// TwinCAT 3 PLC project Untitled1
// ProgramVersion: 3.1.4024.0
// libraries:
//   Tc2_MC2, * (Beckhoff Automation GmbH)
//   Tc2_Standard, * (Beckhoff Automation GmbH)
//   Tc2_System, * (Beckhoff Automation GmbH)
//   Tc3_Module, * (Beckhoff Automation GmbH)
// project tree:
//   GVLs/ GVL_Axes.TcGVL
//   / PlcTask.TcTTO
//   POUs/ MAIN.TcPOU (not stored)
// real-time tasks:
//   TASK PlcTask: cycle T#10ms, priority 20, ADS port 350
// motion (NC):
//   TASK NC-Task 1 SAF: cycle T#2ms, priority 4, ADS port 501
//   TASK NC-Task 1 SVB: cycle T#10ms, priority 8, ADS port 511
//   AXIS Axis 1 (id 1)
//     General: UnitName=Degree
//     OtherSettings: AllowMotionCmdToSlave=true
//     encoder EncType=19
//       EncPara: ScaleFactorNumerator=360, ScaleFactorDenominator=16777216, MaxCount=#xffffffff
//     drive DrvType=16
//       DrvPara: MaxCount=#xffffffff, DriveControlDWord=#x00020000
//         Analog: TorqueSetpointScale=10, ScaleFactorActTorque=0.1
//         TimeComp: TaskDelayCycles=1
//     controller CtrType=1
//       CtrPara: PriorControlFactor=1
//         PosDiffControl: Range=5000
//         Observer: BandWidth=20
//   AXIS Axis 2 (id 2)
//     General: UnitName=Degree
//     OtherSettings: AllowMotionCmdToSlave=true
//     encoder EncType=19
//       EncPara: ScaleFactorNumerator=360, ScaleFactorDenominator=16777216, MaxCount=#xffffffff
//     drive DrvType=16
//       DrvPara: MaxCount=#xffffffff, DriveControlDWord=#x00020000
//         Analog: TorqueSetpointScale=10, ScaleFactorActTorque=0.1
//         TimeComp: TaskDelayCycles=1
//     controller CtrType=1
//       CtrPara: PriorControlFactor=1
//         PosDiffControl: Range=5000
//         Observer: BandWidth=20
//   AXIS Axis 3 (id 3)
//     General: UnitName=Degree
//     OtherSettings: AllowMotionCmdToSlave=true
//     encoder EncType=19
//       EncPara: ScaleFactorNumerator=360, ScaleFactorDenominator=16777216, MaxCount=#xffffffff
//     drive DrvType=16
//       DrvPara: MaxCount=#xffffffff, DriveControlDWord=#x00020000
//         Analog: TorqueSetpointScale=10, ScaleFactorActTorque=0.1
//         TimeComp: TaskDelayCycles=1
//     controller CtrType=1
//       CtrPara: PriorControlFactor=1
//         PosDiffControl: Range=5000
//         Observer: BandWidth=20
//   AXIS Axis 4 (id 4)
//     General: UnitName=Degree
//     OtherSettings: AllowMotionCmdToSlave=true
//     encoder EncType=19
//       EncPara: ScaleFactorNumerator=360, ScaleFactorDenominator=16777216, MaxCount=#xffffffff
//     drive DrvType=16
//       DrvPara: MaxCount=#xffffffff, DriveControlDWord=#x00020000
//         Analog: TorqueSetpointScale=10, ScaleFactorActTorque=0.1
//         TimeComp: TaskDelayCycles=1
//     controller CtrType=1
//       CtrPara: PriorControlFactor=1
//         PosDiffControl: Range=5000
//         Observer: BandWidth=20
//   AXIS Axis 5 (id 5)
//     General: UnitName=Degree
//     OtherSettings: AllowMotionCmdToSlave=true
//     encoder EncType=19
//       EncPara: ScaleFactorNumerator=360, ScaleFactorDenominator=16777216, MaxCount=#xffffffff
//     drive DrvType=16
//       DrvPara: MaxCount=#xffffffff, DriveControlDWord=#x00020000
//         Analog: TorqueSetpointScale=10, ScaleFactorActTorque=0.1
//         TimeComp: TaskDelayCycles=1
//     controller CtrType=1
//       CtrPara: PriorControlFactor=1
//         PosDiffControl: Range=5000
//         Observer: BandWidth=20
//   AXIS Axis 6 (id 6)
//     General: UnitName=Degree
//     OtherSettings: AllowMotionCmdToSlave=true
//     encoder EncType=19
//       EncPara: ScaleFactorNumerator=360, ScaleFactorDenominator=16777216, MaxCount=#xffffffff
//     drive DrvType=16
//       DrvPara: MaxCount=#xffffffff, DriveControlDWord=#x00020000
//         Analog: TorqueSetpointScale=10, ScaleFactorActTorque=0.1
//         TimeComp: TaskDelayCycles=1
//     controller CtrType=1
//       CtrPara: PriorControlFactor=1
//         PosDiffControl: Range=5000
//         Observer: BandWidth=20
// I/O:
//   DEVICE Device 2 (EtherCAT), AmsNetId 169.254.189.18.3.1
//     Drive 1 (SDP-E CoE Drive) [SDP-E CoE Drive]
//     Drive 2 (SDP-E CoE Drive) [SDP-E CoE Drive]
//     Drive 3 (SDP-E CoE Drive) [SDP-E CoE Drive]
//     Drive 4 (SDP-E CoE Drive) [SDP-E CoE Drive]
//     Drive 5 (SDP-E CoE Drive) [SDP-E CoE Drive]
//     Drive 6 (SDP-E CoE Drive) [SDP-E CoE Drive]
// variable links:
//   NC-Task 1 SAF/Axes/Axis 1 <-> Device 2 (EtherCAT)/Drive 1 (SDP-E CoE Drive)
//     Drive/Inputs/In/nDcOutputTime <-> InfoData/DcOutputShift
//     Drive/Inputs/In/nState1 <-> 2nd Transmit PDO Mapping/Statusword
//     Drive/Inputs/In/nState2 <-> 2nd Transmit PDO Mapping/Statusword @bit 8
//     Drive/Inputs/In/nState4 @bit 1 <-> WcState/InputToggle
//     Drive/Inputs/In/nState4 <-> WcState/WcState
//     Drive/Outputs/Out/nCtrl1 <-> 2nd Receive PDO Mapping/Controlword
//     Drive/Outputs/Out/nCtrl2 <-> 2nd Receive PDO Mapping/Controlword @bit 8
//     Drive/Outputs/Out/nDataOut1 <-> 2nd Receive PDO Mapping/Target position
//     Enc/Inputs/In/nDataIn1 <-> 2nd Transmit PDO Mapping/Position actual value
//     Enc/Inputs/In/nDcInputTime <-> InfoData/DcInputShift
//     Enc/Inputs/In/nState4 @bit 1 <-> WcState/InputToggle
//     Enc/Inputs/In/nState4 <-> WcState/WcState
//   NC-Task 1 SAF/Axes/Axis 2 <-> Device 2 (EtherCAT)/Drive 2 (SDP-E CoE Drive)
//     Drive/Inputs/In/nDcOutputTime <-> InfoData/DcOutputShift
//     Drive/Inputs/In/nState1 <-> 2nd Transmit PDO Mapping/Statusword
//     Drive/Inputs/In/nState2 <-> 2nd Transmit PDO Mapping/Statusword @bit 8
//     Drive/Inputs/In/nState4 @bit 1 <-> WcState/InputToggle
//     Drive/Inputs/In/nState4 <-> WcState/WcState
//     Drive/Outputs/Out/nCtrl1 <-> 2nd Receive PDO Mapping/Controlword
//     Drive/Outputs/Out/nCtrl2 <-> 2nd Receive PDO Mapping/Controlword @bit 8
//     Drive/Outputs/Out/nDataOut1 <-> 2nd Receive PDO Mapping/Target position
//     Enc/Inputs/In/nDataIn1 <-> 2nd Transmit PDO Mapping/Position actual value
//     Enc/Inputs/In/nDcInputTime <-> InfoData/DcInputShift
//     Enc/Inputs/In/nState4 @bit 1 <-> WcState/InputToggle
//     Enc/Inputs/In/nState4 <-> WcState/WcState
//   NC-Task 1 SAF/Axes/Axis 3 <-> Device 2 (EtherCAT)/Drive 3 (SDP-E CoE Drive)
//     Drive/Inputs/In/nDcOutputTime <-> InfoData/DcOutputShift
//     Drive/Inputs/In/nState1 <-> 2nd Transmit PDO Mapping/Statusword
//     Drive/Inputs/In/nState2 <-> 2nd Transmit PDO Mapping/Statusword @bit 8
//     Drive/Inputs/In/nState4 @bit 1 <-> WcState/InputToggle
//     Drive/Inputs/In/nState4 <-> WcState/WcState
//     Drive/Outputs/Out/nCtrl1 <-> 2nd Receive PDO Mapping/Controlword
//     Drive/Outputs/Out/nCtrl2 <-> 2nd Receive PDO Mapping/Controlword @bit 8
//     Drive/Outputs/Out/nDataOut1 <-> 2nd Receive PDO Mapping/Target position
//     Enc/Inputs/In/nDataIn1 <-> 2nd Transmit PDO Mapping/Position actual value
//     Enc/Inputs/In/nDcInputTime <-> InfoData/DcInputShift
//     Enc/Inputs/In/nState4 @bit 1 <-> WcState/InputToggle
//     Enc/Inputs/In/nState4 <-> WcState/WcState
//   NC-Task 1 SAF/Axes/Axis 4 <-> Device 2 (EtherCAT)/Drive 4 (SDP-E CoE Drive)
//     Drive/Inputs/In/nDcOutputTime <-> InfoData/DcOutputShift
//     Drive/Inputs/In/nState1 <-> 2nd Transmit PDO Mapping/Statusword
//     Drive/Inputs/In/nState2 <-> 2nd Transmit PDO Mapping/Statusword @bit 8
//     Drive/Inputs/In/nState4 @bit 1 <-> WcState/InputToggle
//     Drive/Inputs/In/nState4 <-> WcState/WcState
//     Drive/Outputs/Out/nCtrl1 <-> 2nd Receive PDO Mapping/Controlword
//     Drive/Outputs/Out/nCtrl2 <-> 2nd Receive PDO Mapping/Controlword @bit 8
//     Drive/Outputs/Out/nDataOut1 <-> 2nd Receive PDO Mapping/Target position
//     Enc/Inputs/In/nDataIn1 <-> 2nd Transmit PDO Mapping/Position actual value
//     Enc/Inputs/In/nDcInputTime <-> InfoData/DcInputShift
//     Enc/Inputs/In/nState4 @bit 1 <-> WcState/InputToggle
//     Enc/Inputs/In/nState4 <-> WcState/WcState
//   NC-Task 1 SAF/Axes/Axis 5 <-> Device 2 (EtherCAT)/Drive 5 (SDP-E CoE Drive)
//     Drive/Inputs/In/nDcOutputTime <-> InfoData/DcOutputShift
//     Drive/Inputs/In/nState1 <-> 2nd Transmit PDO Mapping/Statusword
//     Drive/Inputs/In/nState2 <-> 2nd Transmit PDO Mapping/Statusword @bit 8
//     Drive/Inputs/In/nState4 @bit 1 <-> WcState/InputToggle
//     Drive/Inputs/In/nState4 <-> WcState/WcState
//     Drive/Outputs/Out/nCtrl1 <-> 2nd Receive PDO Mapping/Controlword
//     Drive/Outputs/Out/nCtrl2 <-> 2nd Receive PDO Mapping/Controlword @bit 8
//     Drive/Outputs/Out/nDataOut1 <-> 2nd Receive PDO Mapping/Target position
//     Enc/Inputs/In/nDataIn1 <-> 2nd Transmit PDO Mapping/Position actual value
//     Enc/Inputs/In/nDcInputTime <-> InfoData/DcInputShift
//     Enc/Inputs/In/nState4 @bit 1 <-> WcState/InputToggle
//     Enc/Inputs/In/nState4 <-> WcState/WcState
//   NC-Task 1 SAF/Axes/Axis 6 <-> Device 2 (EtherCAT)/Drive 6 (SDP-E CoE Drive)
//     Drive/Inputs/In/nDcOutputTime <-> InfoData/DcOutputShift
//     Drive/Inputs/In/nState1 <-> 2nd Transmit PDO Mapping/Statusword
//     Drive/Inputs/In/nState2 <-> 2nd Transmit PDO Mapping/Statusword @bit 8
//     Drive/Inputs/In/nState4 @bit 1 <-> WcState/InputToggle
//     Drive/Inputs/In/nState4 <-> WcState/WcState
//     Drive/Outputs/Out/nCtrl1 <-> 2nd Receive PDO Mapping/Controlword
//     Drive/Outputs/Out/nCtrl2 <-> 2nd Receive PDO Mapping/Controlword @bit 8
//     Drive/Outputs/Out/nDataOut1 <-> 2nd Receive PDO Mapping/Target position
//     Enc/Inputs/In/nDataIn1 <-> 2nd Transmit PDO Mapping/Position actual value
//     Enc/Inputs/In/nDcInputTime <-> InfoData/DcInputShift
//     Enc/Inputs/In/nState4 @bit 1 <-> WcState/InputToggle
//     Enc/Inputs/In/nState4 <-> WcState/WcState
//   Untitled1/Untitled1 Instance <-> NC-Task 1 SAF/Axes/Axis 1
//     PlcTask Inputs/GVL_Axes.Axis1.NcToPlc <-> Outputs/ToPlc
//     PlcTask Outputs/GVL_Axes.Axis1.PlcToNc <-> Inputs/FromPlc
//   Untitled1/Untitled1 Instance <-> NC-Task 1 SAF/Axes/Axis 2
//     PlcTask Inputs/GVL_Axes.Axis2.NcToPlc <-> Outputs/ToPlc
//     PlcTask Outputs/GVL_Axes.Axis2.PlcToNc <-> Inputs/FromPlc
//   Untitled1/Untitled1 Instance <-> NC-Task 1 SAF/Axes/Axis 3
//     PlcTask Inputs/GVL_Axes.Axis3.NcToPlc <-> Outputs/ToPlc
//     PlcTask Outputs/GVL_Axes.Axis3.PlcToNc <-> Inputs/FromPlc
//   Untitled1/Untitled1 Instance <-> NC-Task 1 SAF/Axes/Axis 4
//     PlcTask Inputs/GVL_Axes.Axis4.NcToPlc <-> Outputs/ToPlc
//     PlcTask Outputs/GVL_Axes.Axis4.PlcToNc <-> Inputs/FromPlc
//   Untitled1/Untitled1 Instance <-> NC-Task 1 SAF/Axes/Axis 5
//     PlcTask Inputs/GVL_Axes.Axis5.NcToPlc <-> Outputs/ToPlc
//     PlcTask Outputs/GVL_Axes.Axis5.PlcToNc <-> Inputs/FromPlc
//   Untitled1/Untitled1 Instance <-> NC-Task 1 SAF/Axes/Axis 6
//     PlcTask Inputs/GVL_Axes.Axis6.NcToPlc <-> Outputs/ToPlc
//     PlcTask Outputs/GVL_Axes.Axis6.PlcToNc <-> Inputs/FromPlc

CONFIGURATION Untitled1
    RESOURCE PLC ON TwinCAT3
        TASK PlcTask(INTERVAL := T#10ms, PRIORITY := 20);
        PROGRAM MAIN WITH PlcTask : MAIN;
    END_RESOURCE
END_CONFIGURATION

// ---- GVLs/GVL_Axes.TcGVL
VAR_GLOBAL
    Axis1 : AXIS_REF;
    Axis2 : AXIS_REF;
    Axis3 : AXIS_REF;
    Axis4 : AXIS_REF;
    Axis5 : AXIS_REF;
    Axis6 : AXIS_REF;
END_VAR
